{attribute 'OPC.UA.DA' := '1'}
FUNCTION_BLOCK ELL18AttenuationFilter EXTENDS AttenuationFilterBase
VAR_INPUT
END_VAR
VAR_OUTPUT
END_VAR
VAR
	{attribute 'OPC.UA.DA' := '0'}
	_config : ELL18AttenuationFilterConfig;
	{attribute 'OPC.UA.DA' := '0'}
	_coeAccess : CoeAccess;
	{attribute 'OPC.UA.DA' := '0'}
	_initConfigSerialCom : BOOL;	
	{attribute 'OPC.UA.DA' := '0'}
	_serialCom  : SerialCom(Prefix :='', Suffix := Const.CR_LF);
	{attribute 'OPC.UA.DA' := '0'}
	_refSerialCom : REFERENCE TO SerialCom(Prefix :='', Suffix := Const.CR_LF) := _serialCom;	 
	{attribute 'OPC.UA.DA' := '0'}
	_isReceived : BOOL;
	
	{attribute 'OPC.UA.DA' := '0'}
	_deliverMessages : INT;
	
	PositionMsg : STRING(255);
	IdMsg : STRING(255);
	CustomMsg : STRING(255);
	StateMsg : TExecutionState;
	
	{region 'Commands'}	
	
	{attribute 'OPC.UA.DA' := '0'}
	_homePosition 		: BOOL;
	{attribute 'OPC.UA.DA' := '0'}
	_moveAbsPosition    : BOOL;
	{attribute 'OPC.UA.DA' := '0'}
	_moveRelPosition    : BOOL;	
	{attribute 'OPC.UA.DA' := '0'}
	_jogBackwardPosition : BOOL;
	{attribute 'OPC.UA.DA' := '0'}
	_jogForwardPosition  : BOOL;
	{attribute 'OPC.UA.DA' := '0'}
	_customCmd : BOOL;
	{attribute 'OPC.UA.DA' := '0'}			  		   
	_raiseProperties : BOOL;			 
		 
	{endregion}
	
	{attribute 'OPC.UA.DA' := '0'}
	_initDevice : BOOL;	
	 
	{attribute 'OPC.UA.DA' := '0'}
	_pos : LREAL;
	{attribute 'OPC.UA.DA' := '0'}
	_cmd : STRING;	
	{attribute 'OPC.UA.DA' := '0'}
	_itemScheduler : INT;			
	{attribute 'OPC.UA.DA' := '0'}
	_itemRaisedProperties : INT;	
	{attribute 'OPC.UA.DA' := '0'}
	_pulseGenerator : TON;	
			
	{attribute 'OPC.UA.DA' := '0'}
	tmpMessage : STRING;
	{attribute 'OPC.UA.DA' := '0'}
	message : STRING;
	{attribute 'OPC.UA.DA' := '0'}
	_length : INT;		 
	{attribute 'OPC.UA.DA' := '0'}
	_findSuffix : INT;
			
	{attribute 'OPC.UA.DA' := '0'}
	_calibrateStartAngle : LREAL;
	{attribute 'OPC.UA.DA' := '0'}
	_calibrateEndAngle : LREAL;
	{attribute 'OPC.UA.DA' := '0'}
	_angleSteps : LREAL;
	{attribute 'OPC.UA.DA' := '0'}
	_numberAverages : UINT;
	{attribute 'OPC.UA.DA' := '0'}
	_itemCalibrateScheduler : INT;	
	{attribute 'OPC.UA.DA' := '0'}
	_itemPos : UINT;
	{attribute 'OPC.UA.DA' := '0'}
	_pulseCalibration : TON;
		 
	{attribute 'OPC.UA.DA' := '0'}
	PowerMsg : STRING;
		 
	{attribute 'OPC.UA.DA' := '0'}
	_isOpen : BOOL;
	{attribute 'OPC.UA.DA' := '0'}
	_isWriteClose : BOOL;
	{attribute 'OPC.UA.DA' := '0'}
	ValuesCalibrate : ARRAY [0..1000] OF LREAL;
	{attribute 'OPC.UA.DA' := '0'}
	_counter : UINT;
	{attribute 'OPC.UA.DA' := '0'}
	PowerSum : LREAL;
	{attribute 'OPC.UA.DA' := '0'}
	PowerAverage : LREAL;
		 
	{endregion}
	
	{attribute 'OPC.UA.DA' := '0'}
	_lastSetPositionToPulses : DWORD;

	{attribute 'OPC.UA.DA' := '0'}
	InputPiezoBW AT %I* : DINT;
	{attribute 'OPC.UA.DA' := '0'}
	InputPiezoFW AT %I* : DINT;
	{attribute 'OPC.UA.DA' := '0'}
	_rPosition : LREAL; 

END_VAR


IF NOT InitConfigSerialCom THEN
	ConfigureSerialCom();
ELSIF THIS^.Status = TExecutionState.Ready THEN				
	IF _refSerialCom.ErrorReceiveId = COMERROR_NOERROR THEN
		_refSerialCom(TxBuffer:= HardwareGlobalVariables.TxBufferRotatingSwitch, 
		 	      	  RxBuffer:= HardwareGlobalVariables.RxBufferRotatingSwitch);
	END_IF	
				  
	// Init device
	InitDevice(); 				  
				  
	// Deliver messages
	IF _refSerialCom.IsReceived THEN		
		CASE _deliverMessages OF			
			EFeedbackMsgAttenuationELL18.PositionMsg :				
				tmpMessage := DELETE(_refSerialCom.LastReceivedString, 3, 1);
				_length := LEN(tmpMessage);
				_findSuffix := FIND(tmpMessage, Const.CR_LF);
				message := DELETE(tmpMessage, 4, _findSuffix);
				
				PositionMsg := ConvertPulsesToDegrees(message);					    			
			EFeedbackMsgAttenuationELL18.IdMsg :
				IdMsg := _refSerialCom.LastReceivedString;
			EFeedbackMsgAttenuationELL14K.CustomMsg :
				CustomMsg := _refSerialCom.LastReceivedString;						
		END_CASE
	ELSE
		CASE _deliverMessages OF			
			EFeedbackMsgAttenuationELL18.StateMsg :
				StateMsg := State;				
		END_CASE
	END_IF										   	
	
	HomePosition(_homePosition);	
	MoveAbsPosition(_moveAbsPosition, _pos);
	MoveRelPosition(_moveRelPosition, _pos);	
	JogBackwardPosition(_jogBackwardPosition);				
	JogForwardPosition(_jogForwardPosition);
	CustomCommand(_customCmd, _cmd);	
	RaisePropertiesChanged(_raiseProperties);
	
	IF (NOT _homePosition AND NOT _moveAbsPosition AND NOT _moveRelPosition AND NOT _jogBackwardPosition AND NOT _jogForwardPosition 
		AND NOT _customCmd AND NOT _raiseProperties) THEN
		//MessageScheduler();
	END_IF
END_IF

METHOD ConfigureSerialCom
VAR_INPUT
END_VAR
IF _coeAccess.CoeOperation.Ready THEN
	_logger.Information(_message.Reset().Append('Start configuration com serial').ToString());
END_IF;	

_coeAccess.CoeOperation.Start();
_coeAccess(SerialCommunication := _config.SerialCommunication);
	
IF _coeAccess.CoeOperation.Done THEN
	_coeAccess.SetDone();	
 
	_Logger.Information(_message.Reset().
							Append('{').Append(TO_STRING(THIS^.Family)).Append('} : ').
							Append(' - Status : ').Append(TO_STRING(_coeAccess.Status)).ToString());	
	InitConfigSerialCom := TRUE;
END_IF
 
IF _coeAccess.CoeOperation.Error THEN	
	_coeAccess.SetError(0);
	
	_Logger.Error(_message.Reset().
							Append('{').Append(TO_STRING(THIS^.Family)).Append('} : ').
							Append(' - Status : ').Append(TO_STRING(_coeAccess.Status)).ToString());
	InitConfigSerialCom := TRUE;
END_IF

THIS^.Status := _coeAccess.Status;
State := _coeAccess.Status;
END_METHOD

METHOD ConvertDegreesToPulses : STRING
VAR_INPUT
	AnglePosition : LREAL;
END_VAR
VAR
	NumberPulses : DWORD;
	DegreesToPulses : STRING;
END_VAR
NumberPulses := LREAL_TO_DWORD(AnglePosition * Const.PULSES_PER_DEG);	
DegreesToPulses := DWORD_TO_HEXSTR(NumberPulses, 8, FALSE);

_lastSetPositionToPulses := NumberPulses;
ConvertDegreesToPulses := DWORD_TO_HEXSTR(NumberPulses, 8, FALSE );
END_METHOD

METHOD ConvertPulsesToDegrees : STRING;
VAR_INPUT
	Pulses : STRING;
END_VAR
VAR
	pulsesInHex : STRING; 	
	PulsesToDeg : STRING;
	
	pulsesToDowrd : DWORD;
	InterpolationPulsesToDword : DWORD;
	
	gap : INT;
END_VAR
pulsesInHex := CONCAT('16#', Pulses);
pulsesToDowrd := STRING_TO_DWORD(pulsesInHex);

gap := DWORD_TO_INT(_lastSetPositionToPulses) - DWORD_TO_INT(pulsesToDowrd);
(*_logger.Verbose(_message.Reset().Append('gap=').
									 Append(INT_TO_STRING(gap)).ToString());*)

// Interpolation
IF gap > 0 THEN
	InterpolationPulsesToDword := pulsesToDowrd + 1;
ELSIF gap < 0 THEN
	InterpolationPulsesToDword := pulsesToDowrd - 1;	
ELSE
	InterpolationPulsesToDword := pulsesToDowrd;
END_IF

(*_logger.Verbose(_message.Reset().Append(DWORD_TO_STRING(pulsesToDowrd)).Append(';').
									 Append(DWORD_TO_STRING(InterpolationPulsesToDword)).ToString());*)

_rPosition := DWORD_TO_LREAL(InterpolationPulsesToDword) / Const.PULSES_PER_DEG;
PulsesToDeg := LREAL_TO_FMTSTR(_rPosition, 4, TRUE);
ConvertPulsesToDegrees := PulsesToDeg;
END_METHOD

{attribute 'TcRpcEnable' := '1'}
METHOD CustomCommand
VAR_INPUT
	Execute : BOOL;
	Cmd : STRING;
END_VAR
IF Execute THEN
	_logger.Information(_message.Reset().
								Append(_config.Name).
								Append(' - Custom : ').
								Append(Cmd).ToString());
	_deliverMessages := EFeedbackMsgAttenuationELL18.CustomMsg;									
	_serialCom.Send(Cmd);
	
	_customCmd := FALSE;
END_IF
END_METHOD

METHOD FB_init : BOOL
VAR_INPUT
	bInitRetains : BOOL; // if TRUE, the retain variables are initialized (warm start / cold start)
	bInCopyCode : BOOL;  // if TRUE, the instance afterwards gets moved into the copy code (online change)
	Config : ELL18AttenuationFilterConfig;
END_VAR
IF Config.IsEnabled THEN
	_config := Config;
	
	SUPER^._attenuationFilterConfig.Name := Config.Name;
	SUPER^._attenuationFilterConfig.DeviceID := Config.DeviceID;
	SUPER^._attenuationFilterConfig.IsEnabled := Config.IsEnabled;
	SUPER^._attenuationFilterConfig.LogLevel := Config.LogLevel;
	
	SUPER^.Name := Config.Name;
	SUPER^.DeviceID := Config.DeviceID;	
	THIS^.Family := DeviceFamily.AttenuationFilter;
	
	_Logger.Information(_message.Reset().Append('Init ').
							Append('{').Append(TO_STRING(THIS^.Family)).Append('} - ').
							Append('{').Append(TO_STRING(Config.Name)).Append('}').ToString());																													
END_IF
END_METHOD

(** Returns the model number and firmware version **)
METHOD GetIdentifier
VAR_INPUT
END_VAR
VAR
	cmd : STRING := '0i1';
END_VAR
_deliverMessages := EFeedbackMsgAttenuationELL18.IdMsg;	
_serialCom.Send(cmd);
END_METHOD

(** Position Query **)
METHOD PROTECTED GetPosition
VAR_INPUT
END_VAR
VAR
	cmd : STRING := '0gp';
END_VAR
_deliverMessages := EFeedbackMsgAttenuationELL18.PositionMsg;	
_serialCom.Send(cmd);
END_METHOD

{attribute 'TcRpcEnable' := '1'}
METHOD HomePosition
VAR_INPUT
	Execute : BOOL;
END_VAR
VAR
	cmd : STRING := '0ho1';
END_VAR
IF Execute THEN
	_logger.Information(_message.Reset().
								Append(_config.Name).
								Append(' - Home position : ').ToString());
	_serialCom.Send(cmd);
	
	_homePosition := FALSE;
END_IF
END_METHOD

PROPERTY InitConfigSerialCom : BOOL
GET
InitConfigSerialCom := _initConfigSerialCom;
END_GET
SET
_initConfigSerialCom := InitConfigSerialCom;
END_SET
END_PROPERTY

METHOD InitDevice
VAR_INPUT
END_VAR
IF NOT _initDevice THEN	
	_logger.Information(_message.Reset().
								Append(_config.Name).
								Append(' - Init device').ToString());	
	_initDevice := TRUE;	
	
	GetPosition();
END_IF
END_METHOD

{attribute 'TcRpcEnable' := '1'}
METHOD PROTECTED JogBackwardPosition
VAR_INPUT
	Execute : BOOL;
END_VAR
VAR
	cmd : STRING := '0bw';
END_VAR
IF Execute THEN
	_logger.Information(_message.Reset().
								Append(_config.Name).
								Append(' - Jog backward position : ').ToString());
	_serialCom.Send(cmd);
	
	_jogBackwardPosition := FALSE;
END_IF
END_METHOD

{attribute 'TcRpcEnable' := '1'}
METHOD PROTECTED JogForwardPosition
VAR_INPUT
	Execute : BOOL;
END_VAR
VAR
	cmd : STRING := '0fw';
END_VAR
IF Execute THEN
	_logger.Information(_message.Reset().
								Append(_config.Name).
								Append(' - Jog forward position : ').ToString());
	_serialCom.Send(cmd);
	
	_jogForwardPosition := FALSE;
END_IF
END_METHOD

METHOD MessageScheduler
VAR_INPUT
END_VAR
IF _pulseGenerator.Q THEN
	_pulseGenerator(IN := FALSE, PT := T#10MS);
	
	GetPosition();
ELSE
	_pulseGenerator(IN := TRUE, PT := T#100MS);		
END_IF
END_METHOD

{attribute 'TcRpcEnable' := '1'}
METHOD PROTECTED MoveAbsPosition 
VAR_INPUT
	Execute : BOOL;
	Position : LREAL;
END_VAR
VAR
	cmd : STRING := '0ma';
END_VAR
IF Execute THEN
	_pos := Position;	
	_logger.Information(_message.Reset().
								Append(_config.Name).
								Append(' - Move absolute position : ').Append(TO_STRING(_pos)).ToString());
		
	_serialCom.Send(CONCAT(cmd, ConvertDegreesToPulses(_pos)));
	_moveAbsPosition := FALSE;
END_IF
END_METHOD

{attribute 'TcRpcEnable' := '1'}
METHOD PROTECTED MoveRelPosition 
VAR_INPUT
	Execute : BOOL;
	AnglePosition : LREAL;
END_VAR
VAR
	cmd : STRING := '0mr';
END_VAR
IF Execute THEN
	_pos := AnglePosition;
	_logger.Information(_message.Reset().
								Append(_config.Name).
								Append(' - Move relative position : ').Append(TO_STRING(_pos)).ToString());
	
	_serialCom.Send(CONCAT(cmd, ConvertDegreesToPulses(_pos)));	
	_moveRelPosition := FALSE;
END_IF
END_METHOD

{attribute 'TcRpcEnable' := '1'}
METHOD RaisePropertiesChanged
VAR_INPUT
	Execute : BOOL;
END_VAR
IF Execute THEN
	IF THIS^.Status <> TExecutionState.Ready THEN	
		_raiseProperties := FALSE;
		RETURN;
	END_IF	

	_raiseProperties := TRUE;
	
	IF _pulseGenerator.Q THEN
		_pulseGenerator(IN := FALSE, PT := T#10MS);	

		CASE _itemRaisedProperties OF
			0:  StateMsg := TExecutionState.Unknown;
				PositionMsg := ' ';
				IdMsg := ' ';
				CustomMsg := ' ';
				
				_itemRaisedProperties := 10;
			
			10:  GetIdentifier();
				_itemRaisedProperties := 11;
				
			11: _deliverMessages := EFeedbackMsgAttenuationELL18.StateMsg;
				_itemRaisedProperties := 12;
				
			12:  GetPosition();
				_itemRaisedProperties := 13;
			
			13:  _logger.Information(_message.Reset().
								Append(_config.Name).
								Append(' - Attenuation RaisePropertiesChanged').ToString());
				_raiseProperties := FALSE;				
				_itemRaisedProperties := 0;
			
		END_CASE
	ELSE
		_pulseGenerator(IN := TRUE, PT := T#100MS);	
	END_IF
END_IF
END_METHOD

END_FUNCTION_BLOCK

(* stored: Version 1.1.0.1, ProductVersion 3.1.4024.12
   POU ELL18AttenuationFilter: Id {28bacf61-81cd-45b5-9738-5273b7086578}, SpecialFunc None
   Folder Commands: Id {6e891a9f-c25e-4421-9c1a-3ca4a28da60a}
   Method ConfigureSerialCom: Id {e30d1b6e-b434-4fd7-af68-562e802f2214}
   Method ConvertDegreesToPulses: Id {6b1cace6-3fce-42cd-bc21-b7c80f0c5072}
   Method ConvertPulsesToDegrees: Id {86e701e2-3dc4-4d4c-ab10-f00b30234ba5}
   Method CustomCommand: Id {9a7c7b1d-c0fb-47f5-b4aa-a77d7b62f886}
   Method FB_init: Id {267906c3-31cf-4abf-973b-d3794e2a7624}
   Method GetIdentifier: Id {f5ff51d2-37b6-4bc7-8d73-a5214118b6c2}
   Method GetPosition: Id {1fb557fe-7d9e-4a6a-b52b-8c8c6b16b345}
   Method HomePosition: Id {ae6d5b5c-decd-4ede-b8f8-74b4dbec05d1}
   Property InitConfigSerialCom: Id {d3f7c64f-e0fc-4998-92cf-606a48da2b3f}
   Get Get: Id {845aae30-9777-4d1b-a854-0cc67ad67740}
   Set Set: Id {bf294a8a-6625-45d2-a4cf-e0e9bfeddbdf}
   Method InitDevice: Id {06a13da5-22ae-4f58-97f7-cebbb8feaa15}
   Method JogBackwardPosition: Id {7cf0c4ed-0804-4f67-bb2f-7ac7552fccc1}
   Method JogForwardPosition: Id {85f47b87-7109-410b-a0a0-a6ac08901fdb}
   Method MessageScheduler: Id {abf71e7d-fb30-4777-8dc6-d12e22bd3666}
   Method MoveAbsPosition: Id {a4ef234e-5df1-465b-8721-8112f7c31ec3}
   Method MoveRelPosition: Id {26043356-d72e-4f67-8038-371983846d11}
   Method RaisePropertiesChanged: Id {6af4d634-6508-4c56-b4f7-1e526698b33d} *)
